// TIA Portal V17 export
// export: Created 2023-02-14T02:49:10.4517306Z, ExportSetting WithDefaults, DisplayName Totally Integrated Automation Portal, DisplayVersion V17, DisplayName TIA Portal Openness, DisplayVersion V17, DisplayName TIA Portal Teamcenter Gateway, DisplayVersion V17, DisplayName TIA Portal Version Control Interface, DisplayVersion V17, DisplayName SINAMICS Startdrive Advanced, DisplayVersion V17, DisplayName SINAMICS Startdrive G130, G150, S120, S150, SINAMICS MV, S210, DisplayVersion V17, DisplayName SINAMICS Startdrive G110M, G120, G120C, G120D, G120P, G115D, DisplayVersion V17, DisplayName STEP 7 Professional, DisplayVersion V17, DisplayName STEP 7 Safety, DisplayVersion V17, DisplayName WinCC Professional, DisplayVersion V17
FUNCTION_BLOCK "Read FT Comm"   // FB642, LAD
{ S7_Optimized_Access := 'FALSE' }
VERSION : 0.1
// stored: AutoNumber false, IsIECCheckEnabled false, SetENOAutomatically false, UDAEnableTagReadback false
   VAR_INPUT
      Init : Bool;
      Reset : Bool;
      "FT_Vol flow Val" : Real;   // FT_Volume flow Value
      "FT_Vol flow Stat" : Byte;   // FT_Volume flow Status
      "FT_Mass flow Val" : Real;   // FT_Mass flow Value
      "FT_Mass flow Stat" : Byte;   // FT_Mass flow Status
      "FT_Corrected Vol flow Val" : Real;   // FT_Corrected volume flow Value
      "FT_Corrected Vol flow Stat" : Byte;   // FT_Corrected volume flow Status
      "FT_Density Val" : Real;   // FT_Velocity Value
      "FT_Density Stat" : Byte;   // FT_Velocity Status
      "FT_Reference Density Val" : Real;
      "FT_Reference Density Stat" : Byte;
      "FT_Totalizer_1 Val" : Real;   // FT_Totalizer_1 Value
      "FT_Totalizer_1 Stat" : Byte;   // FT_Totalizer_1 Status
      "FT_Totalizer_2 Val" : Real;   // FT_Totalizer_2 Value
      "FT_Totalizer_2 Stat" : Byte;   // FT_Totalizer_2 Status
      "FT_Totalizer_3 Val" : Real;   // FT_Totalizer_3 Value
      "FT_Totalizer_3 Stat" : Byte;   // FT_Totalizer_3 Status
      Instant { ExternalAccessible := 'False'; ExternalVisible := 'False'; ExternalWritable := 'False'} : String;
   END_VAR
   VAR_OUTPUT
      "Q_Vol flow Val" : Real;   // FT_Volume flow Value
      "Q_Vol flow Stat" : Word;   // FT_Volume flow Status
      "Q_Mass flow Val" : Real;   // FT_Mass flow Value
      "Q_Mass flow Stat" : Word;   // FT_Mass flow Status
      "Q_Corrected Vol flow Val" : Real;   // FT_Corrected volume flow Value
      "Q_Corrected Vol flow Stat" : Word;   // FT_Corrected volume flow Status
      "Q_Density Val" : Real;   // FT_Velocity Value
      "Q_Density Stat" : Word;   // FT_Velocity Status
      "Q_Reference Density Val" : Real;
      "Q_Reference Density Stat" : Word;
      "Q_Totalizer_1 Val" : Real;   // FT_Totalizer_1 Value
      "Q_Totalizer_1 Stat" : Word;   // FT_Totalizer_1 Status
      "Q_Totalizer_2 Val" : Real;   // FT_Totalizer_2 Value
      "Q_Totalizer_2 Stat" : Word;   // FT_Totalizer_2 Status
      "Q_Totalizer_3 Val" : Real;   // FT_Totalizer_3 Value
      "Q_Totalizer_3 Stat" : Word;   // FT_Totalizer_3 Status
   END_VAR
   VAR DB_SPECIFIC
      Always_On : Bool;
   END_VAR
BEGIN

REGION Network 1: Aways On
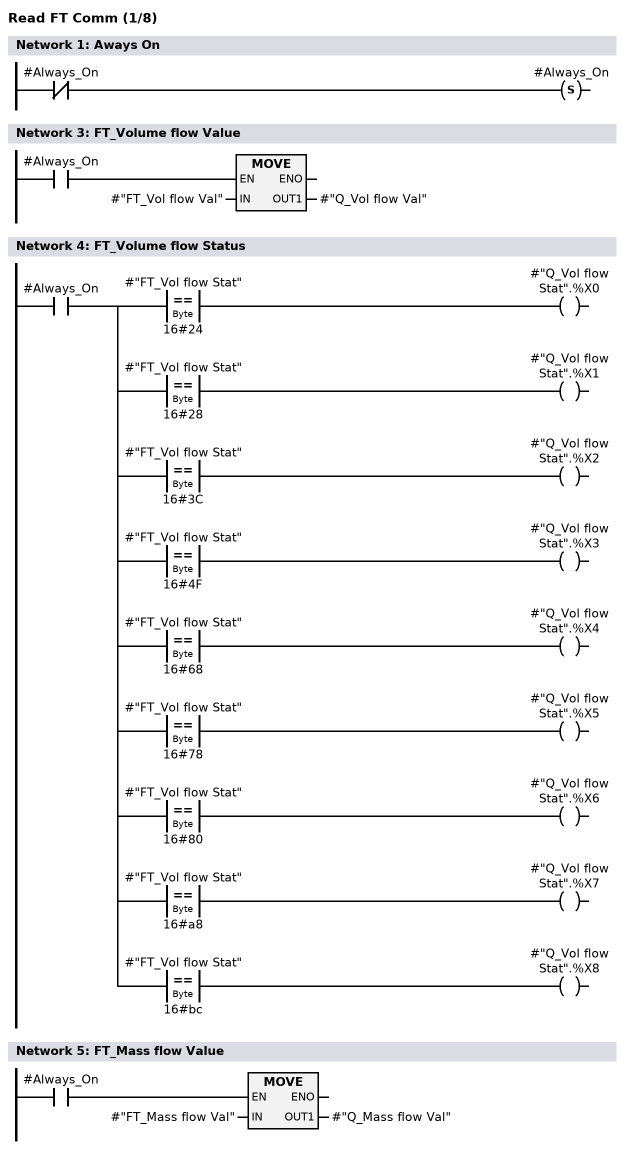
   RUNG wire#powerrail
      I_Contact( #Always_On )
      S_Coil( #Always_On )
   END_RUNG
   // the same network as SCL:
   IF NOT #Always_On THEN #Always_On := TRUE; END_IF;
END_REGION

REGION Network 2: Status Coding
   // 1. 0x24 : BAD - Maintenance alarm - A measured value is not available because a device error has occurred.
   // 2. 0x28 : BAD - Process related - A measured value is not available because the process
   // conditions are not within the device's technical specification limits.
   // 3. 0x3C : BAD - Function check - A function check is active (e.g. cleaning or calibration)
   // 4. 0x4F : UNCERTAIN - Initial value - A pre-defined value is output until a correct measured
   // value is available again or until remedial measures
   // have been carried out that change this status.
   // 5. 0x68 : UNCERTAIN - Maintenance demanded - Signs of wear and tear have been detected on the
   // measuring device. Short-term maintenance is needed to ensure that the measuring device remains
   // operational. The measured value might be invalid. The use of the measured value depends on the application.
   // 6. 0x78 : UNCERTAIN - Process related - The process conditions are not within the device's technical specification limits. This could have a negative impact on the quality and accuracy of the measured value. The use of the measured value depends on the application.
   // 7. 0x80 : GOOD - OK - No error has been diagnosed.
   // 8. 0xA8 : GOOD - Maintenance demanded -  The measured value is valid. It is highly advisable to service the device in the near future.
   // 9. 0xBC :  GOOD - Function check -  The measured value is valid. The measuring device is performing an internal function check. The function check does not have any noticeable effect on the process.
END_REGION

REGION Network 3: FT_Volume flow Value
   RUNG wire#powerrail
      Contact( #Always_On )
      Move(in := #"FT_Vol flow Val", out1 => #"Q_Vol flow Val")
   END_RUNG
   // the same network as SCL:
   IF #Always_On THEN #"Q_Vol flow Val" := #"FT_Vol flow Val"; END_IF;
END_REGION

REGION Network 4: FT_Volume flow Status
   RUNG wire#powerrail
      Contact( #Always_On )
      wire#w1
      { S7_Templates := "SrcType := Byte" } EQ_Contact(in1 := #"FT_Vol flow Stat", in2 := 16#24)
      Coil( #"Q_Vol flow Stat".%X0 )
   END_RUNG
   RUNG wire#w1
      { S7_Templates := "SrcType := Byte" } EQ_Contact(in1 := #"FT_Vol flow Stat", in2 := 16#28)
      Coil( #"Q_Vol flow Stat".%X1 )
   END_RUNG
   RUNG wire#w1
      { S7_Templates := "SrcType := Byte" } EQ_Contact(in1 := #"FT_Vol flow Stat", in2 := 16#3C)
      Coil( #"Q_Vol flow Stat".%X2 )
   END_RUNG
   RUNG wire#w1
      { S7_Templates := "SrcType := Byte" } EQ_Contact(in1 := #"FT_Vol flow Stat", in2 := 16#4F)
      Coil( #"Q_Vol flow Stat".%X3 )
   END_RUNG
   RUNG wire#w1
      { S7_Templates := "SrcType := Byte" } EQ_Contact(in1 := #"FT_Vol flow Stat", in2 := 16#68)
      Coil( #"Q_Vol flow Stat".%X4 )
   END_RUNG
   RUNG wire#w1
      { S7_Templates := "SrcType := Byte" } EQ_Contact(in1 := #"FT_Vol flow Stat", in2 := 16#78)
      Coil( #"Q_Vol flow Stat".%X5 )
   END_RUNG
   RUNG wire#w1
      { S7_Templates := "SrcType := Byte" } EQ_Contact(in1 := #"FT_Vol flow Stat", in2 := 16#80)
      Coil( #"Q_Vol flow Stat".%X6 )
   END_RUNG
   RUNG wire#w1
      { S7_Templates := "SrcType := Byte" } EQ_Contact(in1 := #"FT_Vol flow Stat", in2 := 16#a8)
      Coil( #"Q_Vol flow Stat".%X7 )
   END_RUNG
   RUNG wire#w1
      { S7_Templates := "SrcType := Byte" } EQ_Contact(in1 := #"FT_Vol flow Stat", in2 := 16#bc)
      Coil( #"Q_Vol flow Stat".%X8 )
   END_RUNG
   // the same network as SCL:
   #"Q_Vol flow Stat".%X0 := #Always_On AND (#"FT_Vol flow Stat" = 16#24);
   #"Q_Vol flow Stat".%X1 := #Always_On AND (#"FT_Vol flow Stat" = 16#28);
   #"Q_Vol flow Stat".%X2 := #Always_On AND (#"FT_Vol flow Stat" = 16#3C);
   #"Q_Vol flow Stat".%X3 := #Always_On AND (#"FT_Vol flow Stat" = 16#4F);
   #"Q_Vol flow Stat".%X4 := #Always_On AND (#"FT_Vol flow Stat" = 16#68);
   #"Q_Vol flow Stat".%X5 := #Always_On AND (#"FT_Vol flow Stat" = 16#78);
   #"Q_Vol flow Stat".%X6 := #Always_On AND (#"FT_Vol flow Stat" = 16#80);
   #"Q_Vol flow Stat".%X7 := #Always_On AND (#"FT_Vol flow Stat" = 16#a8);
   #"Q_Vol flow Stat".%X8 := #Always_On AND (#"FT_Vol flow Stat" = 16#bc);
END_REGION

REGION Network 5: FT_Mass flow Value
   RUNG wire#powerrail
      Contact( #Always_On )
      Move(in := #"FT_Mass flow Val", out1 => #"Q_Mass flow Val")
   END_RUNG
   // the same network as SCL:
   IF #Always_On THEN #"Q_Mass flow Val" := #"FT_Mass flow Val"; END_IF;
END_REGION

REGION Network 6: FT_Mass flow Status
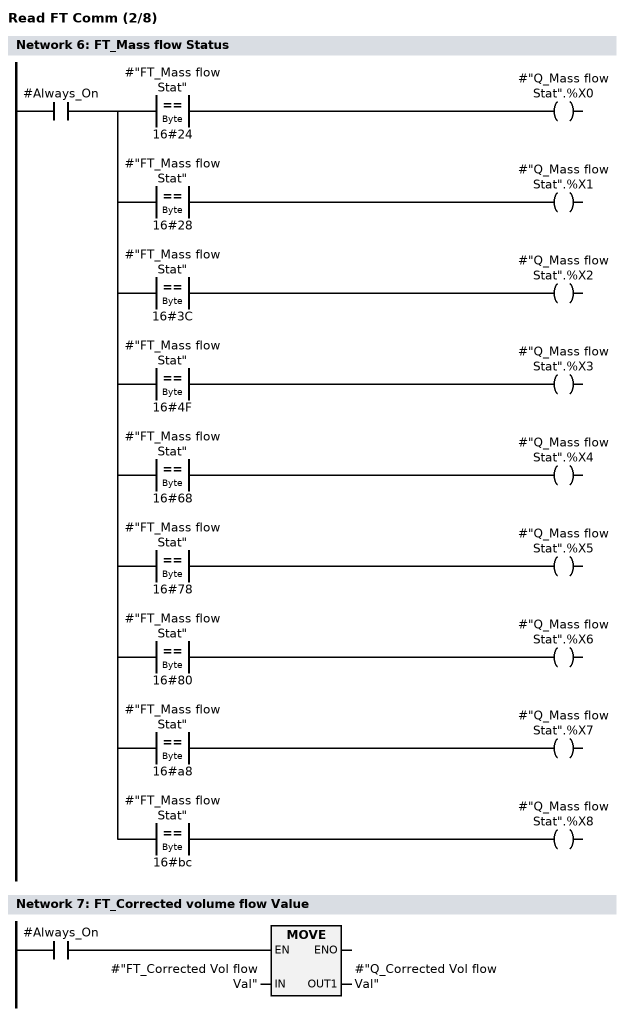
   RUNG wire#powerrail
      Contact( #Always_On )
      wire#w1
      { S7_Templates := "SrcType := Byte" } EQ_Contact(in1 := #"FT_Mass flow Stat", in2 := 16#24)
      Coil( #"Q_Mass flow Stat".%X0 )
   END_RUNG
   RUNG wire#w1
      { S7_Templates := "SrcType := Byte" } EQ_Contact(in1 := #"FT_Mass flow Stat", in2 := 16#28)
      Coil( #"Q_Mass flow Stat".%X1 )
   END_RUNG
   RUNG wire#w1
      { S7_Templates := "SrcType := Byte" } EQ_Contact(in1 := #"FT_Mass flow Stat", in2 := 16#3C)
      Coil( #"Q_Mass flow Stat".%X2 )
   END_RUNG
   RUNG wire#w1
      { S7_Templates := "SrcType := Byte" } EQ_Contact(in1 := #"FT_Mass flow Stat", in2 := 16#4F)
      Coil( #"Q_Mass flow Stat".%X3 )
   END_RUNG
   RUNG wire#w1
      { S7_Templates := "SrcType := Byte" } EQ_Contact(in1 := #"FT_Mass flow Stat", in2 := 16#68)
      Coil( #"Q_Mass flow Stat".%X4 )
   END_RUNG
   RUNG wire#w1
      { S7_Templates := "SrcType := Byte" } EQ_Contact(in1 := #"FT_Mass flow Stat", in2 := 16#78)
      Coil( #"Q_Mass flow Stat".%X5 )
   END_RUNG
   RUNG wire#w1
      { S7_Templates := "SrcType := Byte" } EQ_Contact(in1 := #"FT_Mass flow Stat", in2 := 16#80)
      Coil( #"Q_Mass flow Stat".%X6 )
   END_RUNG
   RUNG wire#w1
      { S7_Templates := "SrcType := Byte" } EQ_Contact(in1 := #"FT_Mass flow Stat", in2 := 16#a8)
      Coil( #"Q_Mass flow Stat".%X7 )
   END_RUNG
   RUNG wire#w1
      { S7_Templates := "SrcType := Byte" } EQ_Contact(in1 := #"FT_Mass flow Stat", in2 := 16#bc)
      Coil( #"Q_Mass flow Stat".%X8 )
   END_RUNG
   // the same network as SCL:
   #"Q_Mass flow Stat".%X0 := #Always_On AND (#"FT_Mass flow Stat" = 16#24);
   #"Q_Mass flow Stat".%X1 := #Always_On AND (#"FT_Mass flow Stat" = 16#28);
   #"Q_Mass flow Stat".%X2 := #Always_On AND (#"FT_Mass flow Stat" = 16#3C);
   #"Q_Mass flow Stat".%X3 := #Always_On AND (#"FT_Mass flow Stat" = 16#4F);
   #"Q_Mass flow Stat".%X4 := #Always_On AND (#"FT_Mass flow Stat" = 16#68);
   #"Q_Mass flow Stat".%X5 := #Always_On AND (#"FT_Mass flow Stat" = 16#78);
   #"Q_Mass flow Stat".%X6 := #Always_On AND (#"FT_Mass flow Stat" = 16#80);
   #"Q_Mass flow Stat".%X7 := #Always_On AND (#"FT_Mass flow Stat" = 16#a8);
   #"Q_Mass flow Stat".%X8 := #Always_On AND (#"FT_Mass flow Stat" = 16#bc);
END_REGION

REGION Network 7: FT_Corrected volume flow Value
   RUNG wire#powerrail
      Contact( #Always_On )
      Move(in := #"FT_Corrected Vol flow Val", out1 => #"Q_Corrected Vol flow Val")
   END_RUNG
   // the same network as SCL:
   IF #Always_On THEN #"Q_Corrected Vol flow Val" := #"FT_Corrected Vol flow Val"; END_IF;
END_REGION

REGION Network 8: FT_Corrected volume flow Status
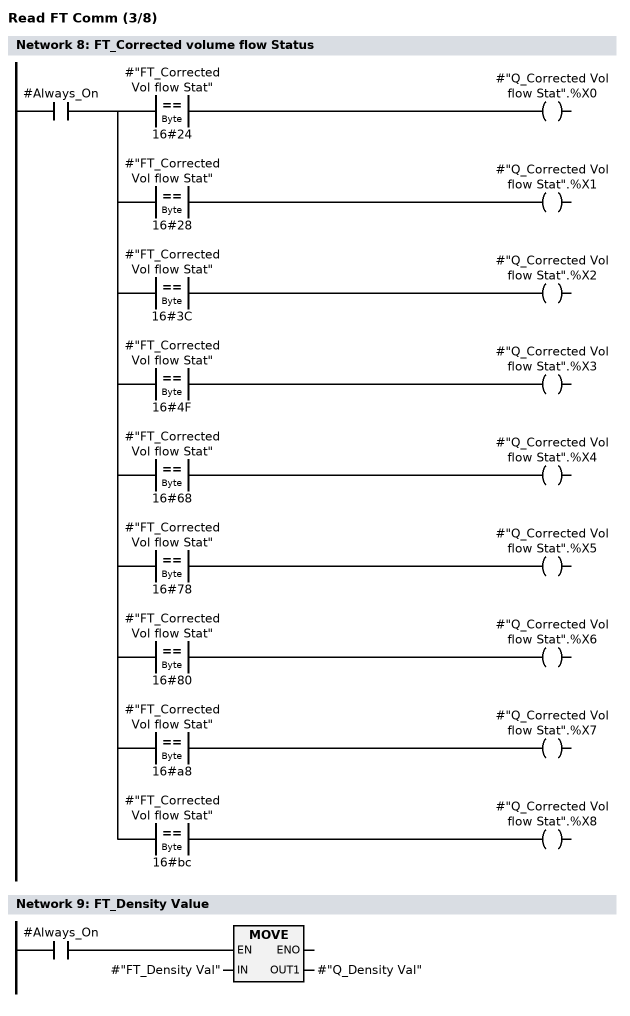
   RUNG wire#powerrail
      Contact( #Always_On )
      wire#w1
      { S7_Templates := "SrcType := Byte" } EQ_Contact(in1 := #"FT_Corrected Vol flow Stat", in2 := 16#24)
      Coil( #"Q_Corrected Vol flow Stat".%X0 )
   END_RUNG
   RUNG wire#w1
      { S7_Templates := "SrcType := Byte" } EQ_Contact(in1 := #"FT_Corrected Vol flow Stat", in2 := 16#28)
      Coil( #"Q_Corrected Vol flow Stat".%X1 )
   END_RUNG
   RUNG wire#w1
      { S7_Templates := "SrcType := Byte" } EQ_Contact(in1 := #"FT_Corrected Vol flow Stat", in2 := 16#3C)
      Coil( #"Q_Corrected Vol flow Stat".%X2 )
   END_RUNG
   RUNG wire#w1
      { S7_Templates := "SrcType := Byte" } EQ_Contact(in1 := #"FT_Corrected Vol flow Stat", in2 := 16#4F)
      Coil( #"Q_Corrected Vol flow Stat".%X3 )
   END_RUNG
   RUNG wire#w1
      { S7_Templates := "SrcType := Byte" } EQ_Contact(in1 := #"FT_Corrected Vol flow Stat", in2 := 16#68)
      Coil( #"Q_Corrected Vol flow Stat".%X4 )
   END_RUNG
   RUNG wire#w1
      { S7_Templates := "SrcType := Byte" } EQ_Contact(in1 := #"FT_Corrected Vol flow Stat", in2 := 16#78)
      Coil( #"Q_Corrected Vol flow Stat".%X5 )
   END_RUNG
   RUNG wire#w1
      { S7_Templates := "SrcType := Byte" } EQ_Contact(in1 := #"FT_Corrected Vol flow Stat", in2 := 16#80)
      Coil( #"Q_Corrected Vol flow Stat".%X6 )
   END_RUNG
   RUNG wire#w1
      { S7_Templates := "SrcType := Byte" } EQ_Contact(in1 := #"FT_Corrected Vol flow Stat", in2 := 16#a8)
      Coil( #"Q_Corrected Vol flow Stat".%X7 )
   END_RUNG
   RUNG wire#w1
      { S7_Templates := "SrcType := Byte" } EQ_Contact(in1 := #"FT_Corrected Vol flow Stat", in2 := 16#bc)
      Coil( #"Q_Corrected Vol flow Stat".%X8 )
   END_RUNG
   // the same network as SCL:
   #"Q_Corrected Vol flow Stat".%X0 := #Always_On AND (#"FT_Corrected Vol flow Stat" = 16#24);
   #"Q_Corrected Vol flow Stat".%X1 := #Always_On AND (#"FT_Corrected Vol flow Stat" = 16#28);
   #"Q_Corrected Vol flow Stat".%X2 := #Always_On AND (#"FT_Corrected Vol flow Stat" = 16#3C);
   #"Q_Corrected Vol flow Stat".%X3 := #Always_On AND (#"FT_Corrected Vol flow Stat" = 16#4F);
   #"Q_Corrected Vol flow Stat".%X4 := #Always_On AND (#"FT_Corrected Vol flow Stat" = 16#68);
   #"Q_Corrected Vol flow Stat".%X5 := #Always_On AND (#"FT_Corrected Vol flow Stat" = 16#78);
   #"Q_Corrected Vol flow Stat".%X6 := #Always_On AND (#"FT_Corrected Vol flow Stat" = 16#80);
   #"Q_Corrected Vol flow Stat".%X7 := #Always_On AND (#"FT_Corrected Vol flow Stat" = 16#a8);
   #"Q_Corrected Vol flow Stat".%X8 := #Always_On AND (#"FT_Corrected Vol flow Stat" = 16#bc);
END_REGION

REGION Network 9: FT_Density Value
   RUNG wire#powerrail
      Contact( #Always_On )
      Move(in := #"FT_Density Val", out1 => #"Q_Density Val")
   END_RUNG
   // the same network as SCL:
   IF #Always_On THEN #"Q_Density Val" := #"FT_Density Val"; END_IF;
END_REGION

REGION Network 10: FT_Density Status
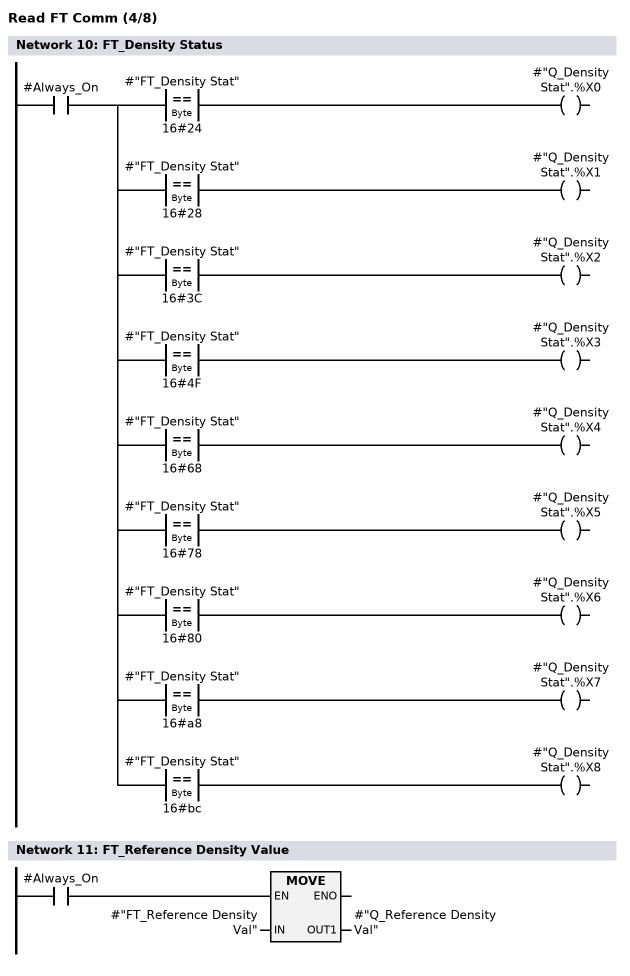
   RUNG wire#powerrail
      Contact( #Always_On )
      wire#w1
      { S7_Templates := "SrcType := Byte" } EQ_Contact(in1 := #"FT_Density Stat", in2 := 16#24)
      Coil( #"Q_Density Stat".%X0 )
   END_RUNG
   RUNG wire#w1
      { S7_Templates := "SrcType := Byte" } EQ_Contact(in1 := #"FT_Density Stat", in2 := 16#28)
      Coil( #"Q_Density Stat".%X1 )
   END_RUNG
   RUNG wire#w1
      { S7_Templates := "SrcType := Byte" } EQ_Contact(in1 := #"FT_Density Stat", in2 := 16#3C)
      Coil( #"Q_Density Stat".%X2 )
   END_RUNG
   RUNG wire#w1
      { S7_Templates := "SrcType := Byte" } EQ_Contact(in1 := #"FT_Density Stat", in2 := 16#4F)
      Coil( #"Q_Density Stat".%X3 )
   END_RUNG
   RUNG wire#w1
      { S7_Templates := "SrcType := Byte" } EQ_Contact(in1 := #"FT_Density Stat", in2 := 16#68)
      Coil( #"Q_Density Stat".%X4 )
   END_RUNG
   RUNG wire#w1
      { S7_Templates := "SrcType := Byte" } EQ_Contact(in1 := #"FT_Density Stat", in2 := 16#78)
      Coil( #"Q_Density Stat".%X5 )
   END_RUNG
   RUNG wire#w1
      { S7_Templates := "SrcType := Byte" } EQ_Contact(in1 := #"FT_Density Stat", in2 := 16#80)
      Coil( #"Q_Density Stat".%X6 )
   END_RUNG
   RUNG wire#w1
      { S7_Templates := "SrcType := Byte" } EQ_Contact(in1 := #"FT_Density Stat", in2 := 16#a8)
      Coil( #"Q_Density Stat".%X7 )
   END_RUNG
   RUNG wire#w1
      { S7_Templates := "SrcType := Byte" } EQ_Contact(in1 := #"FT_Density Stat", in2 := 16#bc)
      Coil( #"Q_Density Stat".%X8 )
   END_RUNG
   // the same network as SCL:
   #"Q_Density Stat".%X0 := #Always_On AND (#"FT_Density Stat" = 16#24);
   #"Q_Density Stat".%X1 := #Always_On AND (#"FT_Density Stat" = 16#28);
   #"Q_Density Stat".%X2 := #Always_On AND (#"FT_Density Stat" = 16#3C);
   #"Q_Density Stat".%X3 := #Always_On AND (#"FT_Density Stat" = 16#4F);
   #"Q_Density Stat".%X4 := #Always_On AND (#"FT_Density Stat" = 16#68);
   #"Q_Density Stat".%X5 := #Always_On AND (#"FT_Density Stat" = 16#78);
   #"Q_Density Stat".%X6 := #Always_On AND (#"FT_Density Stat" = 16#80);
   #"Q_Density Stat".%X7 := #Always_On AND (#"FT_Density Stat" = 16#a8);
   #"Q_Density Stat".%X8 := #Always_On AND (#"FT_Density Stat" = 16#bc);
END_REGION

REGION Network 11: FT_Reference Density Value
   RUNG wire#powerrail
      Contact( #Always_On )
      Move(in := #"FT_Reference Density Val", out1 => #"Q_Reference Density Val")
   END_RUNG
   // the same network as SCL:
   IF #Always_On THEN #"Q_Reference Density Val" := #"FT_Reference Density Val"; END_IF;
END_REGION

REGION Network 12: FT_Reference Density Status
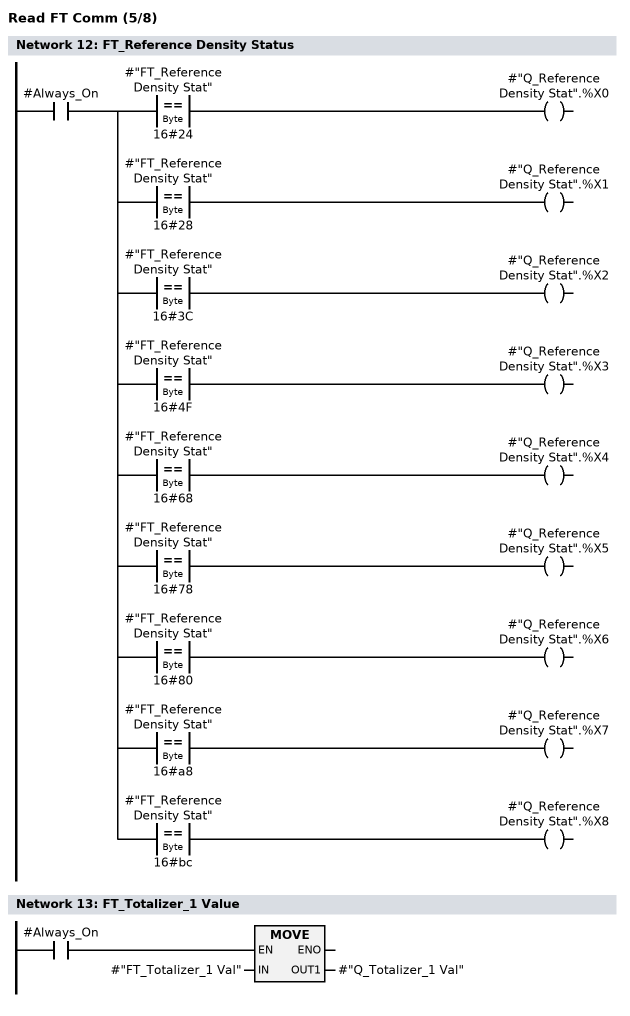
   RUNG wire#powerrail
      Contact( #Always_On )
      wire#w1
      { S7_Templates := "SrcType := Byte" } EQ_Contact(in1 := #"FT_Reference Density Stat", in2 := 16#24)
      Coil( #"Q_Reference Density Stat".%X0 )
   END_RUNG
   RUNG wire#w1
      { S7_Templates := "SrcType := Byte" } EQ_Contact(in1 := #"FT_Reference Density Stat", in2 := 16#28)
      Coil( #"Q_Reference Density Stat".%X1 )
   END_RUNG
   RUNG wire#w1
      { S7_Templates := "SrcType := Byte" } EQ_Contact(in1 := #"FT_Reference Density Stat", in2 := 16#3C)
      Coil( #"Q_Reference Density Stat".%X2 )
   END_RUNG
   RUNG wire#w1
      { S7_Templates := "SrcType := Byte" } EQ_Contact(in1 := #"FT_Reference Density Stat", in2 := 16#4F)
      Coil( #"Q_Reference Density Stat".%X3 )
   END_RUNG
   RUNG wire#w1
      { S7_Templates := "SrcType := Byte" } EQ_Contact(in1 := #"FT_Reference Density Stat", in2 := 16#68)
      Coil( #"Q_Reference Density Stat".%X4 )
   END_RUNG
   RUNG wire#w1
      { S7_Templates := "SrcType := Byte" } EQ_Contact(in1 := #"FT_Reference Density Stat", in2 := 16#78)
      Coil( #"Q_Reference Density Stat".%X5 )
   END_RUNG
   RUNG wire#w1
      { S7_Templates := "SrcType := Byte" } EQ_Contact(in1 := #"FT_Reference Density Stat", in2 := 16#80)
      Coil( #"Q_Reference Density Stat".%X6 )
   END_RUNG
   RUNG wire#w1
      { S7_Templates := "SrcType := Byte" } EQ_Contact(in1 := #"FT_Reference Density Stat", in2 := 16#a8)
      Coil( #"Q_Reference Density Stat".%X7 )
   END_RUNG
   RUNG wire#w1
      { S7_Templates := "SrcType := Byte" } EQ_Contact(in1 := #"FT_Reference Density Stat", in2 := 16#bc)
      Coil( #"Q_Reference Density Stat".%X8 )
   END_RUNG
   // the same network as SCL:
   #"Q_Reference Density Stat".%X0 := #Always_On AND (#"FT_Reference Density Stat" = 16#24);
   #"Q_Reference Density Stat".%X1 := #Always_On AND (#"FT_Reference Density Stat" = 16#28);
   #"Q_Reference Density Stat".%X2 := #Always_On AND (#"FT_Reference Density Stat" = 16#3C);
   #"Q_Reference Density Stat".%X3 := #Always_On AND (#"FT_Reference Density Stat" = 16#4F);
   #"Q_Reference Density Stat".%X4 := #Always_On AND (#"FT_Reference Density Stat" = 16#68);
   #"Q_Reference Density Stat".%X5 := #Always_On AND (#"FT_Reference Density Stat" = 16#78);
   #"Q_Reference Density Stat".%X6 := #Always_On AND (#"FT_Reference Density Stat" = 16#80);
   #"Q_Reference Density Stat".%X7 := #Always_On AND (#"FT_Reference Density Stat" = 16#a8);
   #"Q_Reference Density Stat".%X8 := #Always_On AND (#"FT_Reference Density Stat" = 16#bc);
END_REGION

REGION Network 13: FT_Totalizer_1 Value
   RUNG wire#powerrail
      Contact( #Always_On )
      Move(in := #"FT_Totalizer_1 Val", out1 => #"Q_Totalizer_1 Val")
   END_RUNG
   // the same network as SCL:
   IF #Always_On THEN #"Q_Totalizer_1 Val" := #"FT_Totalizer_1 Val"; END_IF;
END_REGION

REGION Network 14: FT_Totalizer_1 Status
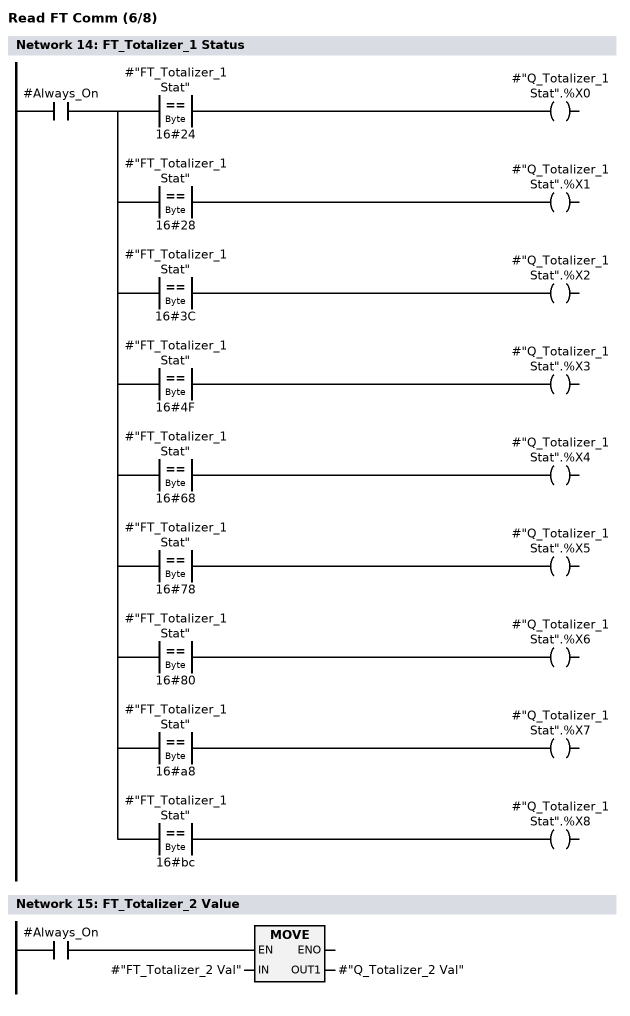
   RUNG wire#powerrail
      Contact( #Always_On )
      wire#w1
      { S7_Templates := "SrcType := Byte" } EQ_Contact(in1 := #"FT_Totalizer_1 Stat", in2 := 16#24)
      Coil( #"Q_Totalizer_1 Stat".%X0 )
   END_RUNG
   RUNG wire#w1
      { S7_Templates := "SrcType := Byte" } EQ_Contact(in1 := #"FT_Totalizer_1 Stat", in2 := 16#28)
      Coil( #"Q_Totalizer_1 Stat".%X1 )
   END_RUNG
   RUNG wire#w1
      { S7_Templates := "SrcType := Byte" } EQ_Contact(in1 := #"FT_Totalizer_1 Stat", in2 := 16#3C)
      Coil( #"Q_Totalizer_1 Stat".%X2 )
   END_RUNG
   RUNG wire#w1
      { S7_Templates := "SrcType := Byte" } EQ_Contact(in1 := #"FT_Totalizer_1 Stat", in2 := 16#4F)
      Coil( #"Q_Totalizer_1 Stat".%X3 )
   END_RUNG
   RUNG wire#w1
      { S7_Templates := "SrcType := Byte" } EQ_Contact(in1 := #"FT_Totalizer_1 Stat", in2 := 16#68)
      Coil( #"Q_Totalizer_1 Stat".%X4 )
   END_RUNG
   RUNG wire#w1
      { S7_Templates := "SrcType := Byte" } EQ_Contact(in1 := #"FT_Totalizer_1 Stat", in2 := 16#78)
      Coil( #"Q_Totalizer_1 Stat".%X5 )
   END_RUNG
   RUNG wire#w1
      { S7_Templates := "SrcType := Byte" } EQ_Contact(in1 := #"FT_Totalizer_1 Stat", in2 := 16#80)
      Coil( #"Q_Totalizer_1 Stat".%X6 )
   END_RUNG
   RUNG wire#w1
      { S7_Templates := "SrcType := Byte" } EQ_Contact(in1 := #"FT_Totalizer_1 Stat", in2 := 16#a8)
      Coil( #"Q_Totalizer_1 Stat".%X7 )
   END_RUNG
   RUNG wire#w1
      { S7_Templates := "SrcType := Byte" } EQ_Contact(in1 := #"FT_Totalizer_1 Stat", in2 := 16#bc)
      Coil( #"Q_Totalizer_1 Stat".%X8 )
   END_RUNG
   // the same network as SCL:
   #"Q_Totalizer_1 Stat".%X0 := #Always_On AND (#"FT_Totalizer_1 Stat" = 16#24);
   #"Q_Totalizer_1 Stat".%X1 := #Always_On AND (#"FT_Totalizer_1 Stat" = 16#28);
   #"Q_Totalizer_1 Stat".%X2 := #Always_On AND (#"FT_Totalizer_1 Stat" = 16#3C);
   #"Q_Totalizer_1 Stat".%X3 := #Always_On AND (#"FT_Totalizer_1 Stat" = 16#4F);
   #"Q_Totalizer_1 Stat".%X4 := #Always_On AND (#"FT_Totalizer_1 Stat" = 16#68);
   #"Q_Totalizer_1 Stat".%X5 := #Always_On AND (#"FT_Totalizer_1 Stat" = 16#78);
   #"Q_Totalizer_1 Stat".%X6 := #Always_On AND (#"FT_Totalizer_1 Stat" = 16#80);
   #"Q_Totalizer_1 Stat".%X7 := #Always_On AND (#"FT_Totalizer_1 Stat" = 16#a8);
   #"Q_Totalizer_1 Stat".%X8 := #Always_On AND (#"FT_Totalizer_1 Stat" = 16#bc);
END_REGION

REGION Network 15: FT_Totalizer_2 Value
   RUNG wire#powerrail
      Contact( #Always_On )
      Move(in := #"FT_Totalizer_2 Val", out1 => #"Q_Totalizer_2 Val")
   END_RUNG
   // the same network as SCL:
   IF #Always_On THEN #"Q_Totalizer_2 Val" := #"FT_Totalizer_2 Val"; END_IF;
END_REGION

REGION Network 16: FT_Totalizer_2 Status
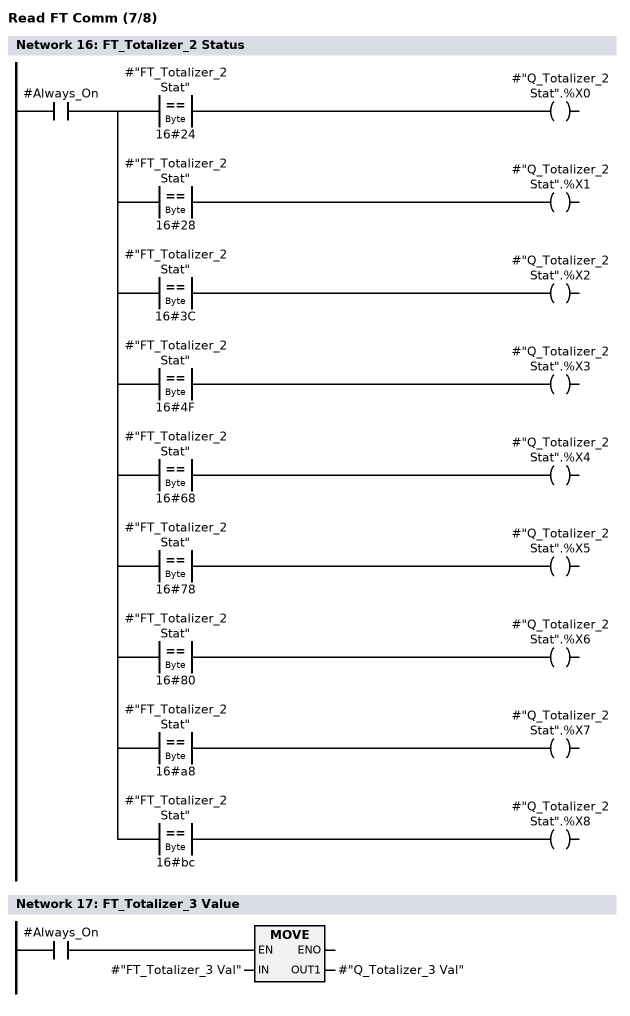
   RUNG wire#powerrail
      Contact( #Always_On )
      wire#w1
      { S7_Templates := "SrcType := Byte" } EQ_Contact(in1 := #"FT_Totalizer_2 Stat", in2 := 16#24)
      Coil( #"Q_Totalizer_2 Stat".%X0 )
   END_RUNG
   RUNG wire#w1
      { S7_Templates := "SrcType := Byte" } EQ_Contact(in1 := #"FT_Totalizer_2 Stat", in2 := 16#28)
      Coil( #"Q_Totalizer_2 Stat".%X1 )
   END_RUNG
   RUNG wire#w1
      { S7_Templates := "SrcType := Byte" } EQ_Contact(in1 := #"FT_Totalizer_2 Stat", in2 := 16#3C)
      Coil( #"Q_Totalizer_2 Stat".%X2 )
   END_RUNG
   RUNG wire#w1
      { S7_Templates := "SrcType := Byte" } EQ_Contact(in1 := #"FT_Totalizer_2 Stat", in2 := 16#4F)
      Coil( #"Q_Totalizer_2 Stat".%X3 )
   END_RUNG
   RUNG wire#w1
      { S7_Templates := "SrcType := Byte" } EQ_Contact(in1 := #"FT_Totalizer_2 Stat", in2 := 16#68)
      Coil( #"Q_Totalizer_2 Stat".%X4 )
   END_RUNG
   RUNG wire#w1
      { S7_Templates := "SrcType := Byte" } EQ_Contact(in1 := #"FT_Totalizer_2 Stat", in2 := 16#78)
      Coil( #"Q_Totalizer_2 Stat".%X5 )
   END_RUNG
   RUNG wire#w1
      { S7_Templates := "SrcType := Byte" } EQ_Contact(in1 := #"FT_Totalizer_2 Stat", in2 := 16#80)
      Coil( #"Q_Totalizer_2 Stat".%X6 )
   END_RUNG
   RUNG wire#w1
      { S7_Templates := "SrcType := Byte" } EQ_Contact(in1 := #"FT_Totalizer_2 Stat", in2 := 16#a8)
      Coil( #"Q_Totalizer_2 Stat".%X7 )
   END_RUNG
   RUNG wire#w1
      { S7_Templates := "SrcType := Byte" } EQ_Contact(in1 := #"FT_Totalizer_2 Stat", in2 := 16#bc)
      Coil( #"Q_Totalizer_2 Stat".%X8 )
   END_RUNG
   // the same network as SCL:
   #"Q_Totalizer_2 Stat".%X0 := #Always_On AND (#"FT_Totalizer_2 Stat" = 16#24);
   #"Q_Totalizer_2 Stat".%X1 := #Always_On AND (#"FT_Totalizer_2 Stat" = 16#28);
   #"Q_Totalizer_2 Stat".%X2 := #Always_On AND (#"FT_Totalizer_2 Stat" = 16#3C);
   #"Q_Totalizer_2 Stat".%X3 := #Always_On AND (#"FT_Totalizer_2 Stat" = 16#4F);
   #"Q_Totalizer_2 Stat".%X4 := #Always_On AND (#"FT_Totalizer_2 Stat" = 16#68);
   #"Q_Totalizer_2 Stat".%X5 := #Always_On AND (#"FT_Totalizer_2 Stat" = 16#78);
   #"Q_Totalizer_2 Stat".%X6 := #Always_On AND (#"FT_Totalizer_2 Stat" = 16#80);
   #"Q_Totalizer_2 Stat".%X7 := #Always_On AND (#"FT_Totalizer_2 Stat" = 16#a8);
   #"Q_Totalizer_2 Stat".%X8 := #Always_On AND (#"FT_Totalizer_2 Stat" = 16#bc);
END_REGION

REGION Network 17: FT_Totalizer_3 Value
   RUNG wire#powerrail
      Contact( #Always_On )
      Move(in := #"FT_Totalizer_3 Val", out1 => #"Q_Totalizer_3 Val")
   END_RUNG
   // the same network as SCL:
   IF #Always_On THEN #"Q_Totalizer_3 Val" := #"FT_Totalizer_3 Val"; END_IF;
END_REGION

REGION Network 18: FT_Totalizer_3 Status
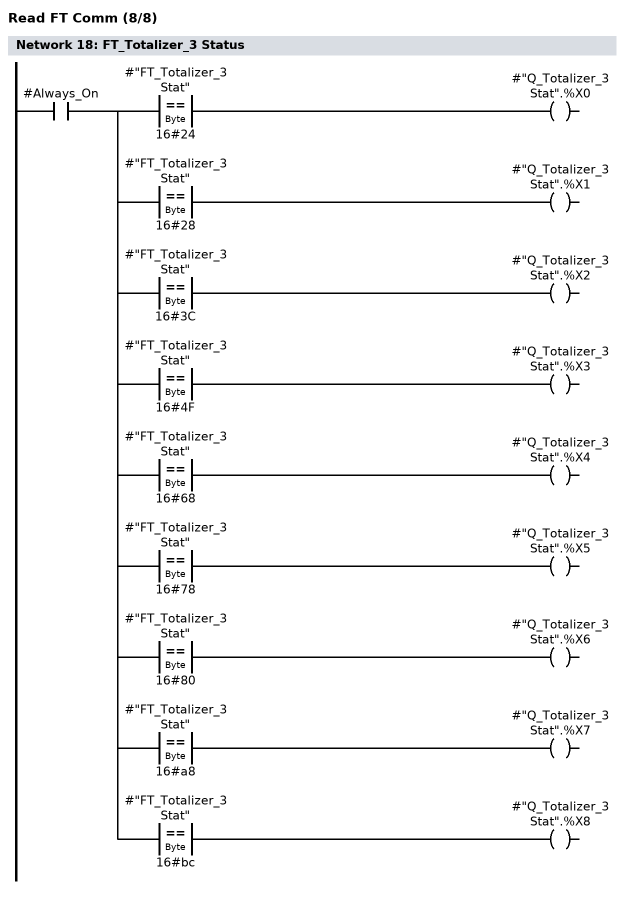
   RUNG wire#powerrail
      Contact( #Always_On )
      wire#w1
      { S7_Templates := "SrcType := Byte" } EQ_Contact(in1 := #"FT_Totalizer_3 Stat", in2 := 16#24)
      Coil( #"Q_Totalizer_3 Stat".%X0 )
   END_RUNG
   RUNG wire#w1
      { S7_Templates := "SrcType := Byte" } EQ_Contact(in1 := #"FT_Totalizer_3 Stat", in2 := 16#28)
      Coil( #"Q_Totalizer_3 Stat".%X1 )
   END_RUNG
   RUNG wire#w1
      { S7_Templates := "SrcType := Byte" } EQ_Contact(in1 := #"FT_Totalizer_3 Stat", in2 := 16#3C)
      Coil( #"Q_Totalizer_3 Stat".%X2 )
   END_RUNG
   RUNG wire#w1
      { S7_Templates := "SrcType := Byte" } EQ_Contact(in1 := #"FT_Totalizer_3 Stat", in2 := 16#4F)
      Coil( #"Q_Totalizer_3 Stat".%X3 )
   END_RUNG
   RUNG wire#w1
      { S7_Templates := "SrcType := Byte" } EQ_Contact(in1 := #"FT_Totalizer_3 Stat", in2 := 16#68)
      Coil( #"Q_Totalizer_3 Stat".%X4 )
   END_RUNG
   RUNG wire#w1
      { S7_Templates := "SrcType := Byte" } EQ_Contact(in1 := #"FT_Totalizer_3 Stat", in2 := 16#78)
      Coil( #"Q_Totalizer_3 Stat".%X5 )
   END_RUNG
   RUNG wire#w1
      { S7_Templates := "SrcType := Byte" } EQ_Contact(in1 := #"FT_Totalizer_3 Stat", in2 := 16#80)
      Coil( #"Q_Totalizer_3 Stat".%X6 )
   END_RUNG
   RUNG wire#w1
      { S7_Templates := "SrcType := Byte" } EQ_Contact(in1 := #"FT_Totalizer_3 Stat", in2 := 16#a8)
      Coil( #"Q_Totalizer_3 Stat".%X7 )
   END_RUNG
   RUNG wire#w1
      { S7_Templates := "SrcType := Byte" } EQ_Contact(in1 := #"FT_Totalizer_3 Stat", in2 := 16#bc)
      Coil( #"Q_Totalizer_3 Stat".%X8 )
   END_RUNG
   // the same network as SCL:
   #"Q_Totalizer_3 Stat".%X0 := #Always_On AND (#"FT_Totalizer_3 Stat" = 16#24);
   #"Q_Totalizer_3 Stat".%X1 := #Always_On AND (#"FT_Totalizer_3 Stat" = 16#28);
   #"Q_Totalizer_3 Stat".%X2 := #Always_On AND (#"FT_Totalizer_3 Stat" = 16#3C);
   #"Q_Totalizer_3 Stat".%X3 := #Always_On AND (#"FT_Totalizer_3 Stat" = 16#4F);
   #"Q_Totalizer_3 Stat".%X4 := #Always_On AND (#"FT_Totalizer_3 Stat" = 16#68);
   #"Q_Totalizer_3 Stat".%X5 := #Always_On AND (#"FT_Totalizer_3 Stat" = 16#78);
   #"Q_Totalizer_3 Stat".%X6 := #Always_On AND (#"FT_Totalizer_3 Stat" = 16#80);
   #"Q_Totalizer_3 Stat".%X7 := #Always_On AND (#"FT_Totalizer_3 Stat" = 16#a8);
   #"Q_Totalizer_3 Stat".%X8 := #Always_On AND (#"FT_Totalizer_3 Stat" = 16#bc);
END_REGION
END_FUNCTION_BLOCK
